// TIA Portal V16 export
// export: Created 2024-09-05T17:36:33.9120078Z, ExportSetting WithDefaults, DisplayName Totally Integrated Automation Portal, DisplayVersion V16 Update 6, DisplayName TIA Portal Version Control Interface, DisplayVersion V16 Update 2, DisplayName TIA Portal Openness, DisplayVersion V16 Update 6, DisplayName STEP 7 Professional, DisplayVersion V16 Update 6, DisplayName STEP 7 Safety, DisplayVersion V16, DisplayName WinCC Advanced, DisplayVersion V16 Update 6
VAR_GLOBAL   // PLC tag table "Cylinders_manual"
   iMM104Wp2__AutoejectGripperLifting AT %I27.2 : Bool;
   iMM350Wp2__ShiftWedgeRight AT %I26.4 : Bool;
   iMM352Wp2__ShiftWedgeLeft AT %I26.7 : Bool;
END_VAR
